(* CODESYS project Industrial module 1.project

Project tree, tasks and I/O mapping:
  CODESYS_Control_for_Raspberry_Pi : CODESYS Control for Raspberry Pi, 3S - Smart Software Solutions GmbH, version 3.5.7.0
    application Application
      task Task (cyclic, interval t#20ms, priority 1) calls POU [Main]
      task VISU_TASK (cyclic, interval 100 ms, priority 31) calls VisuElems.Visu_Prg
      task TrendRecordingTask (cyclic, interval 100 ms, priority 31) calls VisuTrendStorageAccess.GlobalInstances.g_TrendRecordingManager.CyclicCall
      program POU [ST]
      data type AXIS
      visualisation Test_Modbus
      global variables Global
    Onewire
    SPI
    I²C
    GPIOs_A_B : GPIOs A/B, 3S - Smart Software Solutions GmbH, version 1.1.1.0
        unmapped channels: digital inputs (GPIO0..GPIO31), digital outputs (GPIO0..GPIO31)
    SoftMotion General Axis Pool
    Camera device
      <Empty>
    Ethernet : Ethernet, 3S - Smart Software Solutions GmbH, version 3.5.7.0
      Modbus_TCP_Master : Modbus TCP Master, 3S - Smart Software Solutions GmbH, version 3.5.6.0
        Kreativadelar_Modbus_Slave_1 : Modbus TCP Slave, 3S - Smart Software Solutions GmbH, version 3.5.4.0
            settings: Unit-ID = 1; Channel 0.Function Code = 16; Channel 0.Read Offset = 0; Channel 0.Read Length = 0; Channel 0.Write Offset = 16#0008; Channel 0.Write Length = 8; Channel 0.Cycle Time = 100; Channel 1.Function Code = 3; Channel 1.Read Offset = 16#0016; Channel 1.Read Length = 8; Channel 1.Write Offset = 0; Channel 1.Write Length = 0; Channel 1.Cycle Time = 100; Channel 2.Function Code = 15; Channel 2.Read Offset = 0; Channel 2.Read Length = 0; Channel 2.Write Offset = 16#0008; Channel 2.Write Length = 8; Channel 2.Cycle Time = 100; Channel 3.Function Code = 1; Channel 3.Read Offset = 16#0010; Channel 3.Read Length = 8; Channel 3.Write Offset = 0; Channel 3.Write Length = 0; Channel 3.Cycle Time = 100
            output Application.Axis3.Q_Pos : WORD  // Channel 0.Channel 0
            output Application.Axis3.Q_Vel : WORD  // Channel 0.Channel 0
            output Application.Axis3.Q_Acc : WORD  // Channel 0.Channel 0
            output Application.Axis3.Q_Decel : WORD  // Channel 0.Channel 0
            output Application.Axis3.Q_Trans : WORD  // Channel 0.Channel 0
            output Application.Axis3.Q_Home_Off : WORD  // Channel 0.Channel 0
            input  Application.Axis3.I_Pos : WORD  // Channel 1.Channel 1
            input  Application.Axis3.I_Vel : WORD  // Channel 1.Channel 1
            input  Application.Axis3.I_Trans : WORD  // Channel 1.Channel 1
            input  Application.Axis3.I_Home_off : WORD  // Channel 1.Channel 1
            input  Application.Axis3.I_ErrorId : WORD  // Channel 1.Channel 1
            output Application.Axis3.Q_Exec : BOOL  // Channel 2.Channel 2.Bit0
            output Application.Axis3.Q_Reset : BOOL  // Channel 2.Channel 2.Bit1
            output Application.Axis3.Q_Mode : BOOL  // Channel 2.Channel 2.Bit2
            output Application.Axis3.Q_Forw : BOOL  // Channel 2.Channel 2.Bit3
            output Application.Axis3.Q_Stop : BOOL  // Channel 2.Channel 2.Bit4
            output Application.Axis3.Q_Rev : BOOL  // Channel 2.Channel 2.Bit5
            output Application.Axis3.Q_Homing : BOOL  // Channel 2.Channel 2.Bit6
            output Application.Axis3.Q_Auto_Homing : BOOL  // Channel 2.Channel 2.Bit7
            input  Application.Axis3.I_Ready : BOOL  // Channel 3.Channel 3.Bit0
            input  Application.Axis3.I_Busy : BOOL  // Channel 3.Channel 3.Bit1
            input  Application.Axis3.I_Stop : BOOL  // Channel 3.Channel 3.Bit2
            input  Application.Axis3.I_Pos_Done : BOOL  // Channel 3.Channel 3.Bit3
            input  Application.Axis3.I_Home : BOOL  // Channel 3.Channel 3.Bit4
            input  Application.Axis3.I_Mode : BOOL  // Channel 3.Channel 3.Bit5
            input  Application.Axis3.I_Error : BOOL  // Channel 3.Channel 3.Bit6
            unmapped channels: Channel 0, Channel 1, Channel 2, Channel 3
  text list GlobalTextList
*)

// CODESYS_Control_for_Raspberry_Pi/Application/AXIS
TYPE AXIS :
STRUCT

	Q_Pos : WORD;
	Q_Vel : WORD;
	Q_Acc : WORD;
	Q_Decel : WORD; 
	Q_Trans : WORD;
	Q_Home_Off : WORD;

	Q_Exec : BOOL;
	Q_Reset : BOOL;
	Q_Mode : BOOL;
	Q_Forw : BOOL;
	Q_Stop : BOOL;
	Q_Rev : BOOL;
	Q_Homing : BOOL;
	Q_Auto_Homing : BOOL;

	I_Pos : WORD;
	I_Vel : WORD;
	I_Trans : WORD;
	I_Home_off : WORD;
	I_ErrorId : WORD;
	
	I_Ready : BOOL;
	I_Busy : BOOL;
	I_Stop : BOOL;
	I_Pos_Done : BOOL;
	I_Home : BOOL;
	I_Mode : BOOL;
	I_Error : BOOL;

END_STRUCT
END_TYPE

// CODESYS_Control_for_Raspberry_Pi/Application/Global
VAR_GLOBAL
	Axis3 : AXIS;
END_VAR

// CODESYS_Control_for_Raspberry_Pi/Application/POU
PROGRAM POU
VAR
END_VAR

END_PROGRAM

// CODESYS_Control_for_Raspberry_Pi/Application/Test_Modbus
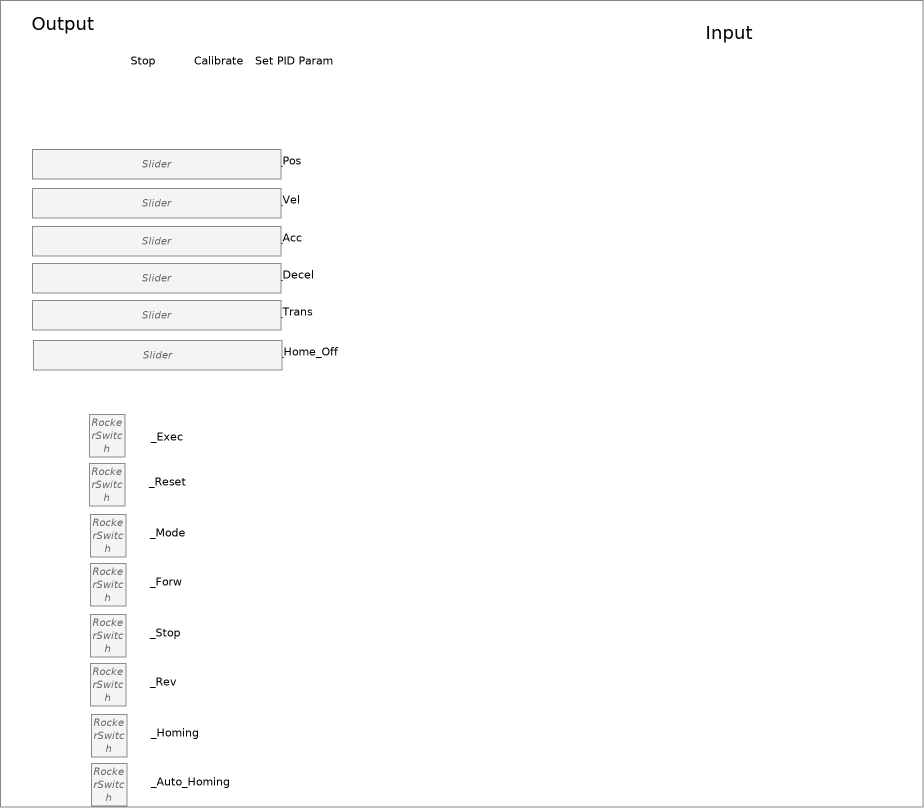
VISUALIZATION Test_Modbus  // 924x808
    Label (-12,9 150x30), "Output"
    Label (654,18 150x30), "Input"
    Label (274,146 150x30), "_Pos"
    Label (68,46 150x30), "Stop"
    Label (144,46 150x30), "Calibrate"
    Label (219,46 150x30), "Set PID Param"
    Label (772,97 150x30)
    RockerSwitch (89,414 36x43), variable: Axis3.Q_Exec, behaviour: TOGGLE, style: Switch-RockerSwitch-Gray
    Label (146,467 150x30), "_Reset"
    RockerSwitch (89,463 36x43), variable: Axis3.Q_Exec, behaviour: TOGGLE, style: Switch-RockerSwitch-Gray
    Label (147,518 150x30), "_Mode"
    RockerSwitch (90,514 36x43), variable: Axis3.Q_Exec, behaviour: TOGGLE, style: Switch-RockerSwitch-Gray
    Label (147,567 150x30), "_Forw"
    RockerSwitch (90,563 36x43), variable: Axis3.Q_Exec, behaviour: TOGGLE, style: Switch-RockerSwitch-Gray
    Label (147,618 150x30), "_Stop"
    RockerSwitch (90,614 36x43), variable: Axis3.Q_Exec, behaviour: TOGGLE, style: Switch-RockerSwitch-Gray
    Label (147,667 150x30), "_Rev"
    RockerSwitch (90,663 36x43), variable: Axis3.Q_Exec, behaviour: TOGGLE, style: Switch-RockerSwitch-Gray
    Label (148,718 150x30), "_Homing"
    RockerSwitch (91,714 36x43), variable: Axis3.Q_Exec, behaviour: TOGGLE, style: Switch-RockerSwitch-Gray
    Label (148,767 150x30), "_Auto_Homing"
    RockerSwitch (91,763 36x43), variable: Axis3.Q_Exec, behaviour: TOGGLE, style: Switch-RockerSwitch-Gray
    Slider (32,149 249x30), scale 0..100
    Label (274,185 150x30), "_Vel"
    Slider (32,188 249x30), scale 0..100
    Label (274,223 150x30), "_Acc"
    Slider (32,226 249x30), scale 0..100
    Label (274,260 150x30), "_Decel"
    Slider (32,263 249x30), scale 0..100
    Label (274,297 150x30), "_Trans"
    Slider (32,300 249x30), scale 0..100
    Label (148,422 150x30), "_Exec"
    Label (275,337 150x30), "_Home_Off"
    Slider (33,340 249x30), scale 0..100
END_VISUALIZATION
